(* CoDeSys 2.3.9.62 project: Tema1 DepositoDosNiveles v0.pro *)

(* Global variable list: Global_Variables *)
VAR_GLOBAL

  (* Variables de entrada *)
  N1:BOOL;
  N2:BOOL;
  N3:BOOL;
  M :BOOL;
  Nivel:BOOL;
  (*Variables de salida *)
  BLLenado:BOOL;
  BVaciado:BOOL;
  LuzN1:BOOL;
  LuzN2:BOOL;
  LuzSubida:BOOL;
END_VAR

(* POU PLC_PRG, ST *)
PROGRAM PLC_PRG
VAR
  posy:INT;

	Desague: BOOL;
END_VAR
Control();


IF BLlenado=TRUE THEN
IF posy>-187 THEN
  posy:=posy-1;
END_IF
END_IF

IF BVaciado=TRUE THEN
IF posy<52 THEN
  posy:=posy+1;
END_IF
END_IF



IF posy<-121 THEN
  N2:=TRUE;
ELSE
  N2:=FALSE;
END_IF

IF posy<-166 THEN
  N1:=TRUE;
ELSE
  N1:=FALSE;
END_IF

IF posy<-10 THEN
  N3:=TRUE;
ELSE
  N3:=FALSE;
END_IF
END_PROGRAM

(* POU Control, LD *)
PROGRAM Control
VAR

	NAux: BOOL;
END_VAR
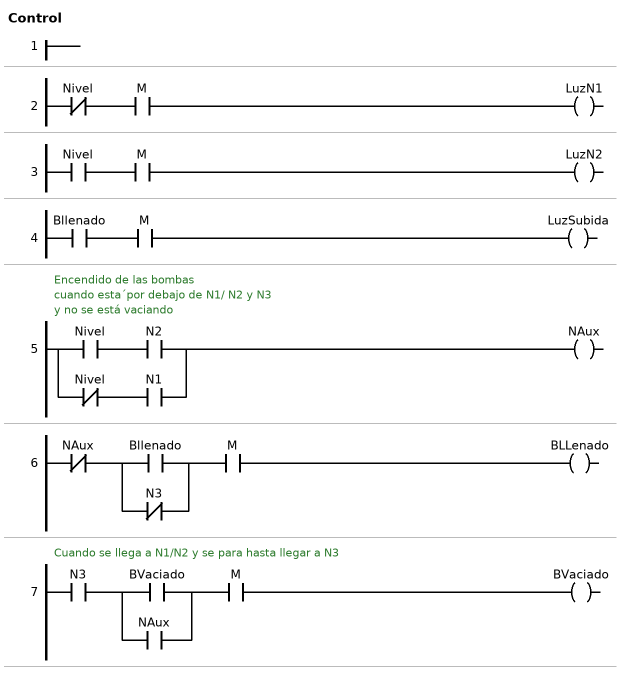
_LD_ (* Ladder Diagram *)
NETWORK 1
	*
NETWORK 2
	[/Nivel] - [M] --- (LuzN1)
NETWORK 3
	[Nivel] - [M] --- (LuzN2)
NETWORK 4
	[Bllenado] - [M] --- (LuzSubida)
NETWORK 5 (* Encendido de las bombas / cuando esta´por debajo de N1/ N2 y N3 / y no se está vaciando *)
	{ [Nivel] - [N2] | [/Nivel] - [N1] } --- (NAux)
NETWORK 6
	[/NAux] - { [Bllenado] | [/N3] } - [M] --- (BLLenado)
NETWORK 7 (* Cuando se llega a N1/N2 y se para hasta llegar a N3 *)
	[N3] - { [BVaciado] | [NAux] } - [M] --- (BVaciado)
_END_LD_
(* the same logic as Structured Text *)
(* Network 1 *)
(* Network 2 *)
LuzN1 := NOT Nivel AND M;
(* Network 3 *)
LuzN2 := Nivel AND M;
(* Network 4 *)
LuzSubida := Bllenado AND M;
(* Network 5: Encendido de las bombas / cuando esta´por debajo de N1/ N2 y N3 / y no se está vaciando *)
NAux := Nivel AND N2 OR NOT Nivel AND N1;
(* Network 6 *)
BLLenado := NOT NAux AND (Bllenado OR NOT N3) AND M;
(* Network 7: Cuando se llega a N1/N2 y se para hasta llegar a N3 *)
BVaciado := N3 AND (BVaciado OR NAux) AND M;
END_PROGRAM

(* Visualisation Deposito
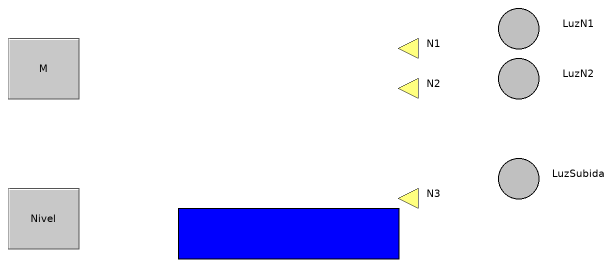
button at (50,80)-(121,141): text "M"; toggles M
polygon at (440,80)-(460,100): alarm colour if .N1; toggles .N1
polygon at (440,120)-(460,140): alarm colour if .N2; toggles .N2
rectangle at (460,70)-(491,101): text "N1"
rectangle at (460,110)-(491,141): text "N2"
rectangle at (220,250)-(441,301): top PLC_PRG.posy
polygon at (440,230)-(460,250): alarm colour if .N3; toggles .N3
button at (50,230)-(121,291): text "Nivel"; toggles Nivel
rectangle at (460,220)-(491,251): text "N3"
ellipse at (540,50)-(581,91): alarm colour if LuzN1
ellipse at (540,100)-(581,141): alarm colour if LuzN2
rectangle at (590,50)-(651,81): text "LuzN1"
rectangle at (590,100)-(651,131): text "LuzN2"
ellipse at (540,200)-(581,241): alarm colour if LuzSubida
rectangle at (590,200)-(651,231): text "LuzSubida"
1 more shapes without text or variables
*)
